PROGRAM AxisVertMovementOutputCtrl_Arm1
VAR
	VertTop: CMP_OC_DW;

	LdVertdown: CMP_OC_DW;
	Stn1Vertdown: CMP_OC_DW;
	Stn2Vertdown: CMP_OC_DW;
	Stn3Vertdown: CMP_OC_DW;
	Stn4Vertdown: CMP_OC_DW;
	Stn5Vertdown: CMP_OC_DW;
	Stn6Vertdown: CMP_OC_DW;
	Stn7Vertdown: CMP_OC_DW;
	Stn8Vertdown: CMP_OC_DW;
	Stn9Vertdown: CMP_OC_DW;
	Stn10Vertdown: CMP_OC_DW;
	Stn11Vertdown: CMP_OC_DW;
	Stn12Vertdown: CMP_OC_DW;
	Uld1Vertdown: CMP_OC_DW;
	Uld2Vertdown: CMP_OC_DW;

	Stn8VertSlowPulldown: CMP_OC_DW;

	Stn9VertSlowPulldown: CMP_OC_DW;
END_VAR

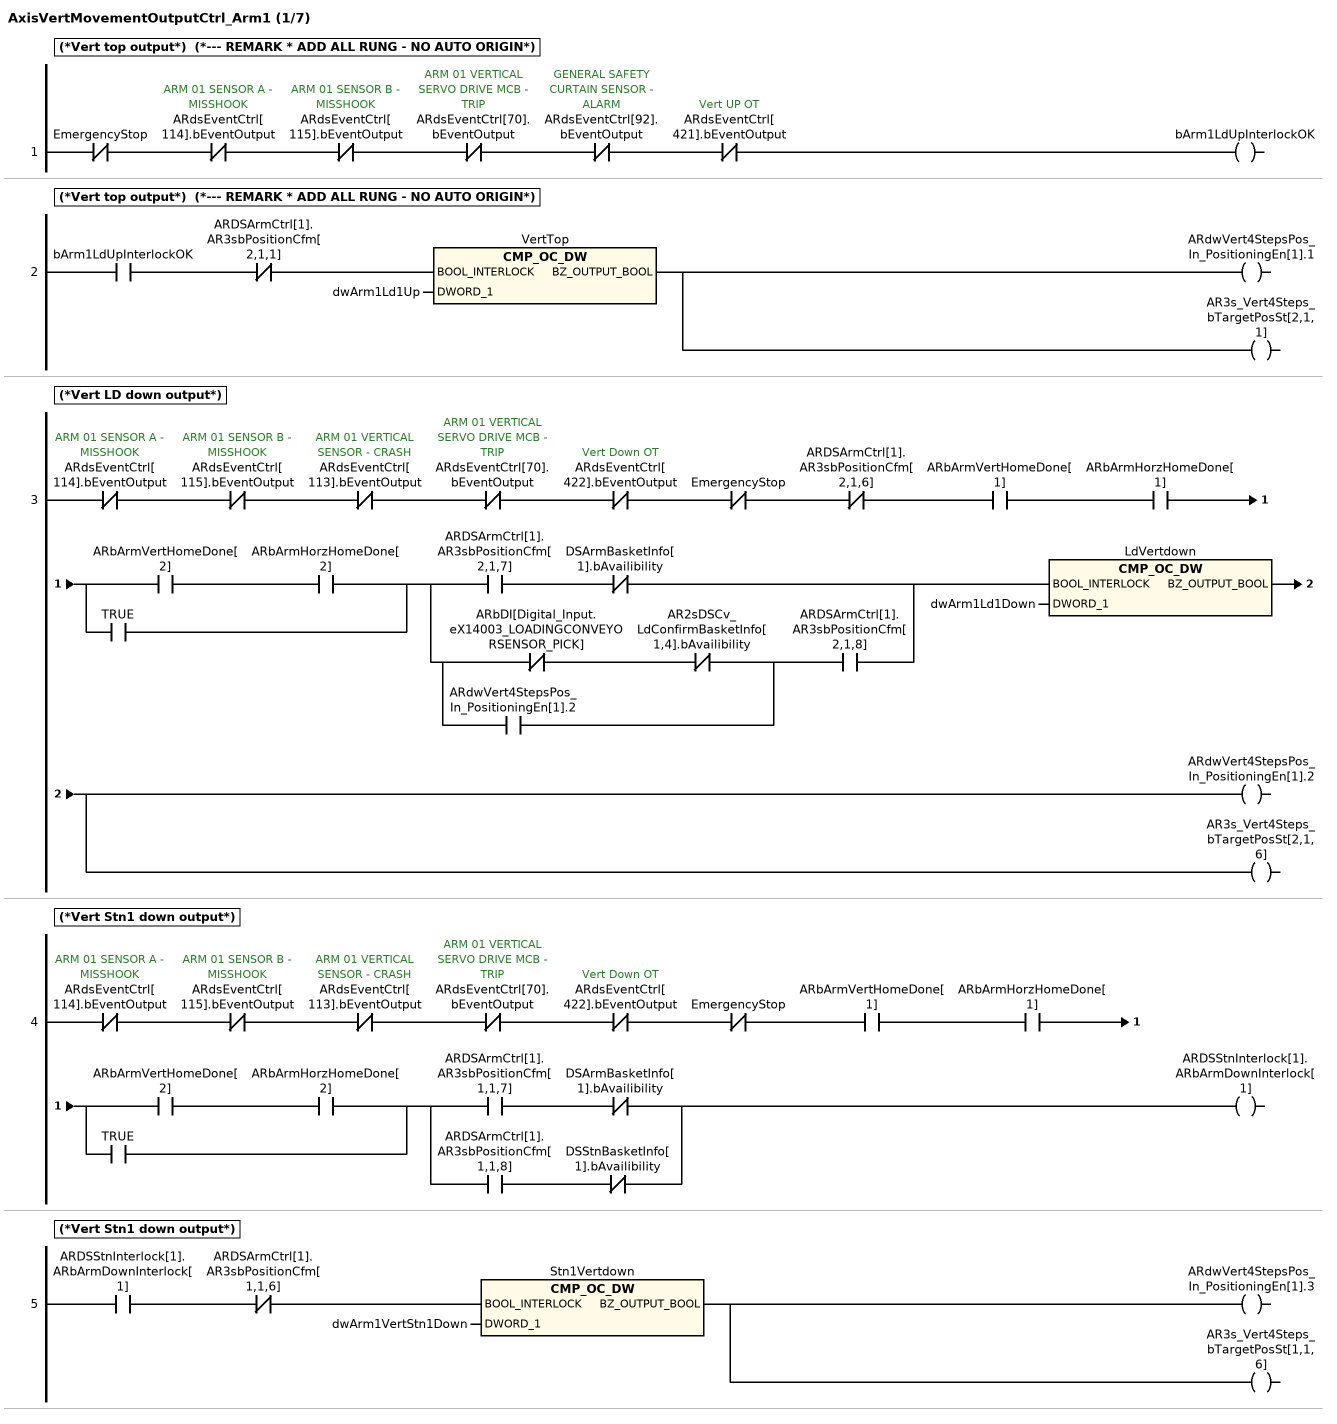
// NETWORK 1
//   ARdsEventCtrl[114].bEventOutput: ARM 01 SENSOR A - MISSHOOK
//   ARdsEventCtrl[115].bEventOutput: ARM 01 SENSOR B - MISSHOOK
//   ARdsEventCtrl[70].bEventOutput: ARM 01 VERTICAL SERVO DRIVE MCB - TRIP
//   ARdsEventCtrl[92].bEventOutput: GENERAL SAFETY CURTAIN SENSOR - ALARM
//   ARdsEventCtrl[421].bEventOutput: Vert UP OT
// label: (*Vert top output*)  (*--- REMARK * ADD ALL RUNG - NO AUTO ORIGIN*)
bArm1LdUpInterlockOK := NOT EmergencyStop AND NOT ARdsEventCtrl[114].bEventOutput AND NOT ARdsEventCtrl[115].bEventOutput AND NOT ARdsEventCtrl[70].bEventOutput AND NOT ARdsEventCtrl[92].bEventOutput AND NOT ARdsEventCtrl[421].bEventOutput;

// NETWORK 2
// label: (*Vert top output*)  (*--- REMARK * ADD ALL RUNG - NO AUTO ORIGIN*)
VertTop(BOOL_INTERLOCK := bArm1LdUpInterlockOK AND NOT ARDSArmCtrl[1].AR3sbPositionCfm[2,1,1], DWORD_1 := dwArm1Ld1Up); // CMP_OC_DW
ARdwVert4StepsPos_In_PositioningEn[1].1 := VertTop.BZ_OUTPUT_BOOL;
AR3s_Vert4Steps_bTargetPosSt[2,1,1] := VertTop.BZ_OUTPUT_BOOL;

// NETWORK 3
//   ARdsEventCtrl[114].bEventOutput: ARM 01 SENSOR A - MISSHOOK
//   ARdsEventCtrl[115].bEventOutput: ARM 01 SENSOR B - MISSHOOK
//   ARdsEventCtrl[113].bEventOutput: ARM 01 VERTICAL SENSOR - CRASH
//   ARdsEventCtrl[70].bEventOutput: ARM 01 VERTICAL SERVO DRIVE MCB - TRIP
//   ARdsEventCtrl[422].bEventOutput: Vert Down OT
// label: (*Vert LD down output*)
LdVertdown(BOOL_INTERLOCK := (NOT ARdsEventCtrl[114].bEventOutput AND NOT ARdsEventCtrl[115].bEventOutput AND NOT ARdsEventCtrl[113].bEventOutput AND NOT ARdsEventCtrl[70].bEventOutput AND NOT ARdsEventCtrl[422].bEventOutput AND NOT EmergencyStop) AND NOT ARDSArmCtrl[1].AR3sbPositionCfm[2,1,6] AND ARbArmVertHomeDone[1] AND ARbArmHorzHomeDone[1] AND (ARbArmVertHomeDone[2] AND ARbArmHorzHomeDone[2] OR TRUE) AND (ARDSArmCtrl[1].AR3sbPositionCfm[2,1,7] AND NOT DSArmBasketInfo[1].bAvailibility OR (NOT ARbDI[Digital_Input.eX14003_LOADINGCONVEYORSENSOR_PICK] AND NOT AR2sDSCv_LdConfirmBasketInfo[1,4].bAvailibility OR ARdwVert4StepsPos_In_PositioningEn[1].2) AND ARDSArmCtrl[1].AR3sbPositionCfm[2,1,8]), DWORD_1 := dwArm1Ld1Down); // CMP_OC_DW
ARdwVert4StepsPos_In_PositioningEn[1].2 := LdVertdown.BZ_OUTPUT_BOOL;
AR3s_Vert4Steps_bTargetPosSt[2,1,6] := LdVertdown.BZ_OUTPUT_BOOL;

// NETWORK 4
//   ARdsEventCtrl[114].bEventOutput: ARM 01 SENSOR A - MISSHOOK
//   ARdsEventCtrl[115].bEventOutput: ARM 01 SENSOR B - MISSHOOK
//   ARdsEventCtrl[113].bEventOutput: ARM 01 VERTICAL SENSOR - CRASH
//   ARdsEventCtrl[70].bEventOutput: ARM 01 VERTICAL SERVO DRIVE MCB - TRIP
//   ARdsEventCtrl[422].bEventOutput: Vert Down OT
// label: (*Vert Stn1 down output*)
ARDSStnInterlock[1].ARbArmDownInterlock[1] := (NOT ARdsEventCtrl[114].bEventOutput AND NOT ARdsEventCtrl[115].bEventOutput AND NOT ARdsEventCtrl[113].bEventOutput AND NOT ARdsEventCtrl[70].bEventOutput AND NOT ARdsEventCtrl[422].bEventOutput AND NOT EmergencyStop) AND ARbArmVertHomeDone[1] AND ARbArmHorzHomeDone[1] AND (ARbArmVertHomeDone[2] AND ARbArmHorzHomeDone[2] OR TRUE) AND (ARDSArmCtrl[1].AR3sbPositionCfm[1,1,7] AND NOT DSArmBasketInfo[1].bAvailibility OR ARDSArmCtrl[1].AR3sbPositionCfm[1,1,8] AND NOT DSStnBasketInfo[1].bAvailibility);

// NETWORK 5
// label: (*Vert Stn1 down output*)
Stn1Vertdown(BOOL_INTERLOCK := ARDSStnInterlock[1].ARbArmDownInterlock[1] AND NOT ARDSArmCtrl[1].AR3sbPositionCfm[1,1,6], DWORD_1 := dwArm1VertStn1Down); // CMP_OC_DW
ARdwVert4StepsPos_In_PositioningEn[1].3 := Stn1Vertdown.BZ_OUTPUT_BOOL;
AR3s_Vert4Steps_bTargetPosSt[1,1,6] := Stn1Vertdown.BZ_OUTPUT_BOOL;

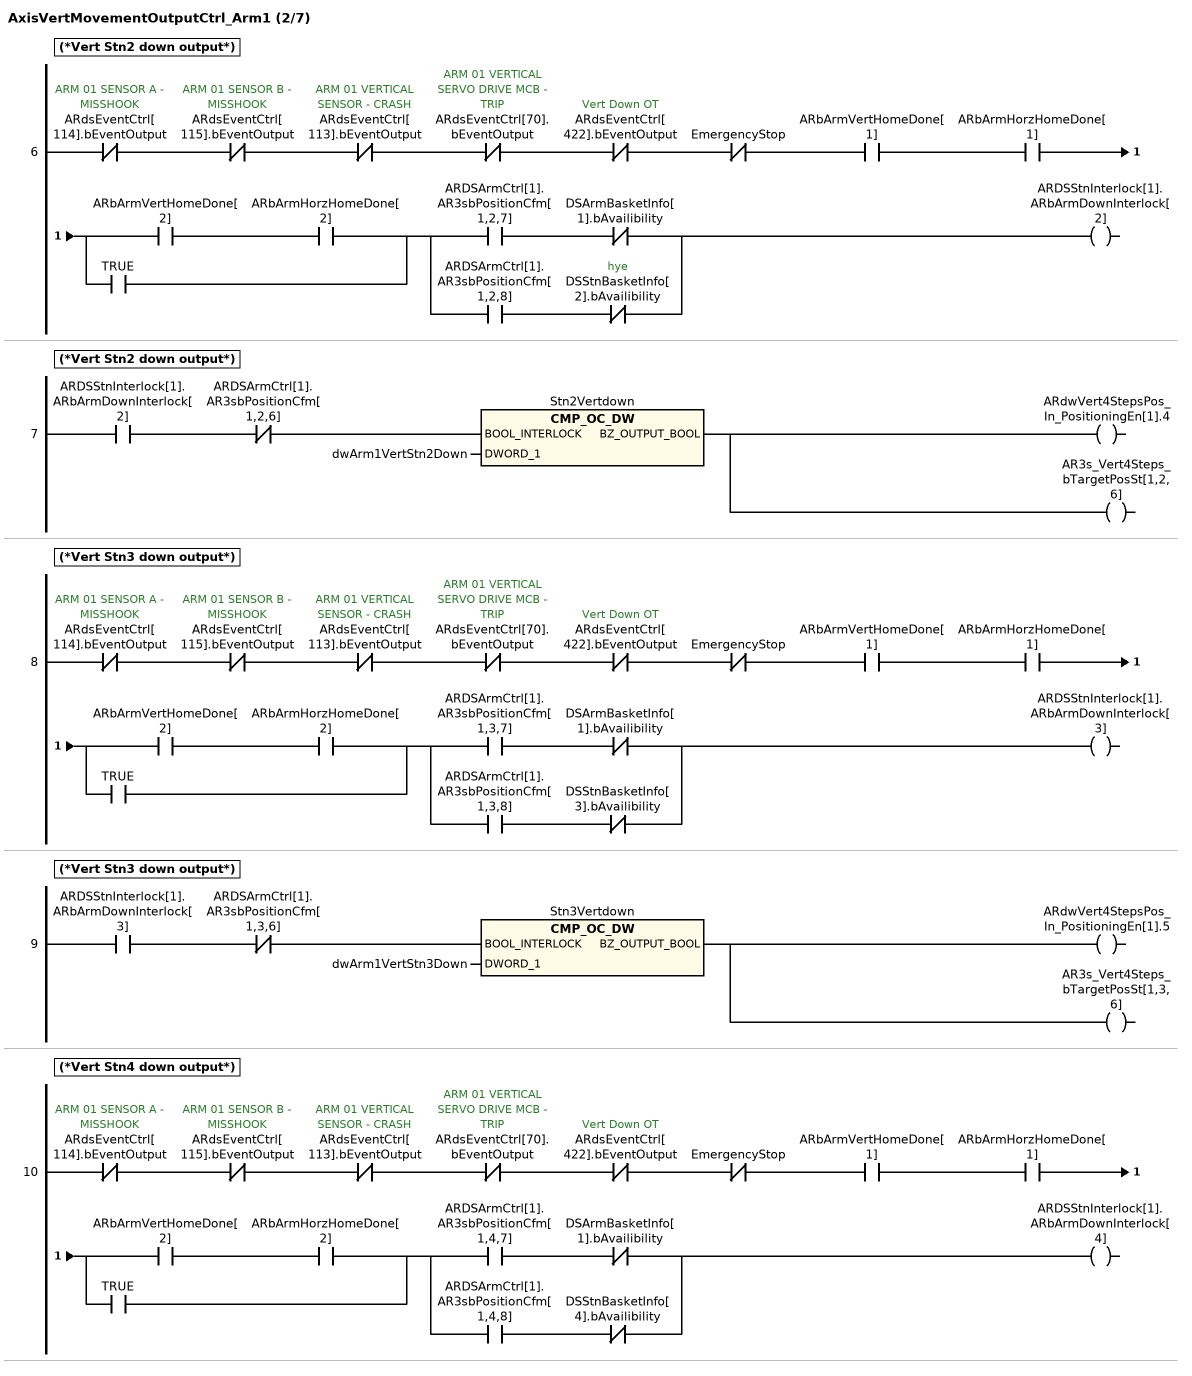
// NETWORK 6
//   ARdsEventCtrl[114].bEventOutput: ARM 01 SENSOR A - MISSHOOK
//   ARdsEventCtrl[115].bEventOutput: ARM 01 SENSOR B - MISSHOOK
//   ARdsEventCtrl[113].bEventOutput: ARM 01 VERTICAL SENSOR - CRASH
//   ARdsEventCtrl[70].bEventOutput: ARM 01 VERTICAL SERVO DRIVE MCB - TRIP
//   ARdsEventCtrl[422].bEventOutput: Vert Down OT
//   DSStnBasketInfo[2].bAvailibility: hye
// label: (*Vert Stn2 down output*)
ARDSStnInterlock[1].ARbArmDownInterlock[2] := (NOT ARdsEventCtrl[114].bEventOutput AND NOT ARdsEventCtrl[115].bEventOutput AND NOT ARdsEventCtrl[113].bEventOutput AND NOT ARdsEventCtrl[70].bEventOutput AND NOT ARdsEventCtrl[422].bEventOutput AND NOT EmergencyStop) AND ARbArmVertHomeDone[1] AND ARbArmHorzHomeDone[1] AND (ARbArmVertHomeDone[2] AND ARbArmHorzHomeDone[2] OR TRUE) AND (ARDSArmCtrl[1].AR3sbPositionCfm[1,2,7] AND NOT DSArmBasketInfo[1].bAvailibility OR ARDSArmCtrl[1].AR3sbPositionCfm[1,2,8] AND NOT DSStnBasketInfo[2].bAvailibility);

// NETWORK 7
// label: (*Vert Stn2 down output*)
Stn2Vertdown(BOOL_INTERLOCK := ARDSStnInterlock[1].ARbArmDownInterlock[2] AND NOT ARDSArmCtrl[1].AR3sbPositionCfm[1,2,6], DWORD_1 := dwArm1VertStn2Down); // CMP_OC_DW
ARdwVert4StepsPos_In_PositioningEn[1].4 := Stn2Vertdown.BZ_OUTPUT_BOOL;
AR3s_Vert4Steps_bTargetPosSt[1,2,6] := Stn2Vertdown.BZ_OUTPUT_BOOL;

// NETWORK 8
//   ARdsEventCtrl[114].bEventOutput: ARM 01 SENSOR A - MISSHOOK
//   ARdsEventCtrl[115].bEventOutput: ARM 01 SENSOR B - MISSHOOK
//   ARdsEventCtrl[113].bEventOutput: ARM 01 VERTICAL SENSOR - CRASH
//   ARdsEventCtrl[70].bEventOutput: ARM 01 VERTICAL SERVO DRIVE MCB - TRIP
//   ARdsEventCtrl[422].bEventOutput: Vert Down OT
// label: (*Vert Stn3 down output*)
ARDSStnInterlock[1].ARbArmDownInterlock[3] := (NOT ARdsEventCtrl[114].bEventOutput AND NOT ARdsEventCtrl[115].bEventOutput AND NOT ARdsEventCtrl[113].bEventOutput AND NOT ARdsEventCtrl[70].bEventOutput AND NOT ARdsEventCtrl[422].bEventOutput AND NOT EmergencyStop) AND ARbArmVertHomeDone[1] AND ARbArmHorzHomeDone[1] AND (ARbArmVertHomeDone[2] AND ARbArmHorzHomeDone[2] OR TRUE) AND (ARDSArmCtrl[1].AR3sbPositionCfm[1,3,7] AND NOT DSArmBasketInfo[1].bAvailibility OR ARDSArmCtrl[1].AR3sbPositionCfm[1,3,8] AND NOT DSStnBasketInfo[3].bAvailibility);

// NETWORK 9
// label: (*Vert Stn3 down output*)
Stn3Vertdown(BOOL_INTERLOCK := ARDSStnInterlock[1].ARbArmDownInterlock[3] AND NOT ARDSArmCtrl[1].AR3sbPositionCfm[1,3,6], DWORD_1 := dwArm1VertStn3Down); // CMP_OC_DW
ARdwVert4StepsPos_In_PositioningEn[1].5 := Stn3Vertdown.BZ_OUTPUT_BOOL;
AR3s_Vert4Steps_bTargetPosSt[1,3,6] := Stn3Vertdown.BZ_OUTPUT_BOOL;

// NETWORK 10
//   ARdsEventCtrl[114].bEventOutput: ARM 01 SENSOR A - MISSHOOK
//   ARdsEventCtrl[115].bEventOutput: ARM 01 SENSOR B - MISSHOOK
//   ARdsEventCtrl[113].bEventOutput: ARM 01 VERTICAL SENSOR - CRASH
//   ARdsEventCtrl[70].bEventOutput: ARM 01 VERTICAL SERVO DRIVE MCB - TRIP
//   ARdsEventCtrl[422].bEventOutput: Vert Down OT
// label: (*Vert Stn4 down output*)
ARDSStnInterlock[1].ARbArmDownInterlock[4] := (NOT ARdsEventCtrl[114].bEventOutput AND NOT ARdsEventCtrl[115].bEventOutput AND NOT ARdsEventCtrl[113].bEventOutput AND NOT ARdsEventCtrl[70].bEventOutput AND NOT ARdsEventCtrl[422].bEventOutput AND NOT EmergencyStop) AND ARbArmVertHomeDone[1] AND ARbArmHorzHomeDone[1] AND (ARbArmVertHomeDone[2] AND ARbArmHorzHomeDone[2] OR TRUE) AND (ARDSArmCtrl[1].AR3sbPositionCfm[1,4,7] AND NOT DSArmBasketInfo[1].bAvailibility OR ARDSArmCtrl[1].AR3sbPositionCfm[1,4,8] AND NOT DSStnBasketInfo[4].bAvailibility);

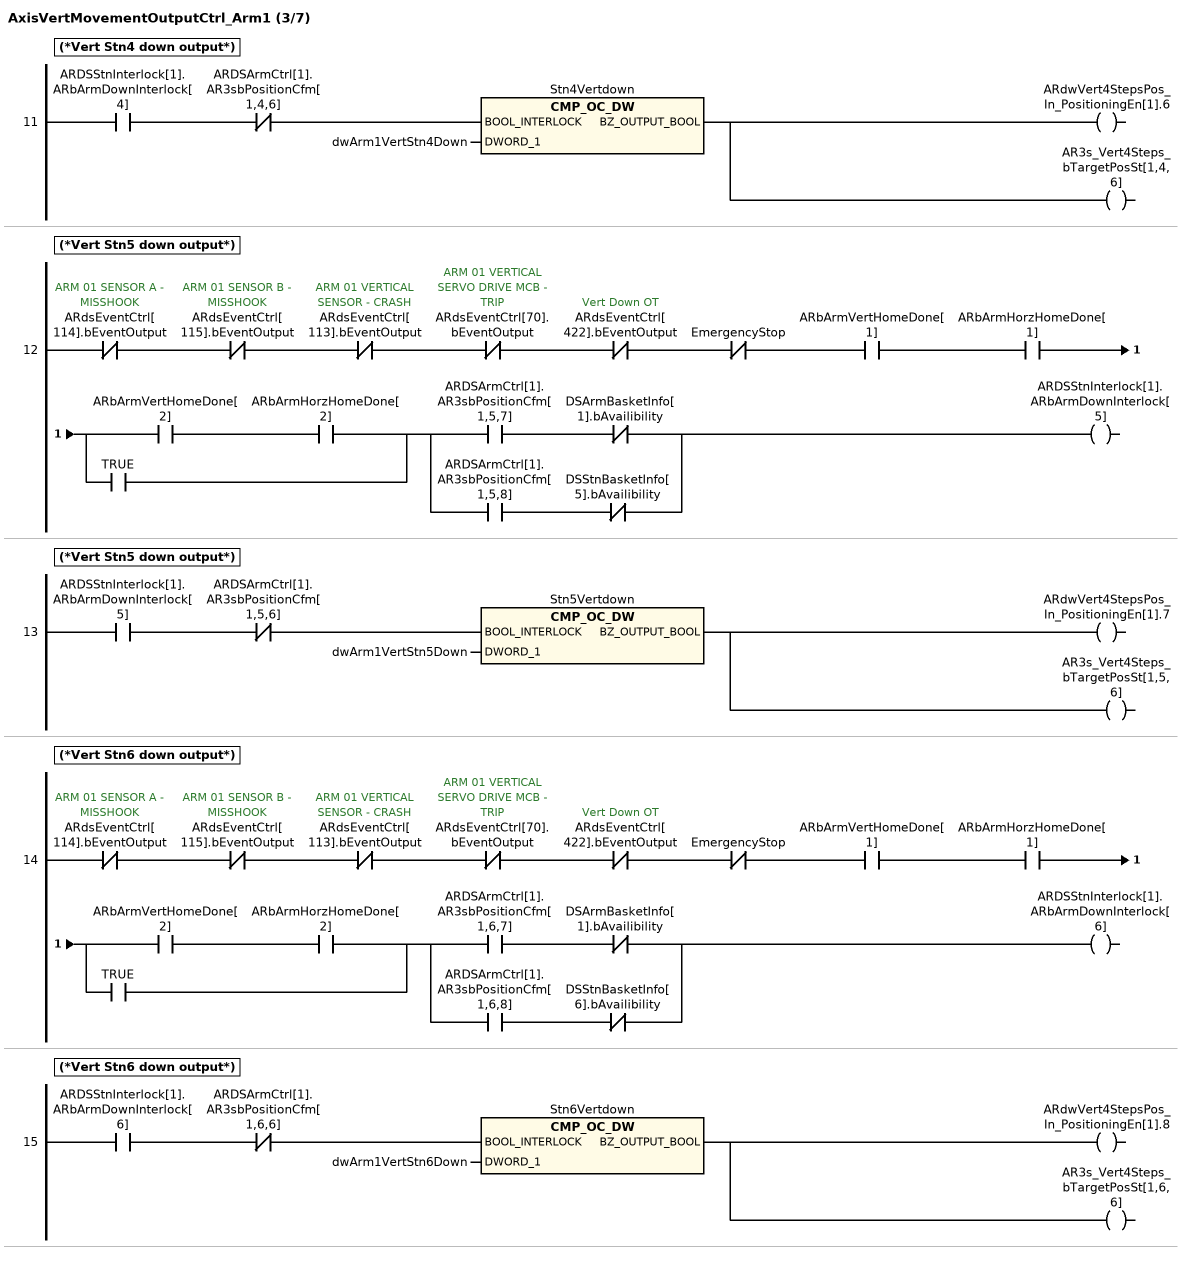
// NETWORK 11
// label: (*Vert Stn4 down output*)
Stn4Vertdown(BOOL_INTERLOCK := ARDSStnInterlock[1].ARbArmDownInterlock[4] AND NOT ARDSArmCtrl[1].AR3sbPositionCfm[1,4,6], DWORD_1 := dwArm1VertStn4Down); // CMP_OC_DW
ARdwVert4StepsPos_In_PositioningEn[1].6 := Stn4Vertdown.BZ_OUTPUT_BOOL;
AR3s_Vert4Steps_bTargetPosSt[1,4,6] := Stn4Vertdown.BZ_OUTPUT_BOOL;

// NETWORK 12
//   ARdsEventCtrl[114].bEventOutput: ARM 01 SENSOR A - MISSHOOK
//   ARdsEventCtrl[115].bEventOutput: ARM 01 SENSOR B - MISSHOOK
//   ARdsEventCtrl[113].bEventOutput: ARM 01 VERTICAL SENSOR - CRASH
//   ARdsEventCtrl[70].bEventOutput: ARM 01 VERTICAL SERVO DRIVE MCB - TRIP
//   ARdsEventCtrl[422].bEventOutput: Vert Down OT
// label: (*Vert Stn5 down output*)
ARDSStnInterlock[1].ARbArmDownInterlock[5] := (NOT ARdsEventCtrl[114].bEventOutput AND NOT ARdsEventCtrl[115].bEventOutput AND NOT ARdsEventCtrl[113].bEventOutput AND NOT ARdsEventCtrl[70].bEventOutput AND NOT ARdsEventCtrl[422].bEventOutput AND NOT EmergencyStop) AND ARbArmVertHomeDone[1] AND ARbArmHorzHomeDone[1] AND (ARbArmVertHomeDone[2] AND ARbArmHorzHomeDone[2] OR TRUE) AND (ARDSArmCtrl[1].AR3sbPositionCfm[1,5,7] AND NOT DSArmBasketInfo[1].bAvailibility OR ARDSArmCtrl[1].AR3sbPositionCfm[1,5,8] AND NOT DSStnBasketInfo[5].bAvailibility);

// NETWORK 13
// label: (*Vert Stn5 down output*)
Stn5Vertdown(BOOL_INTERLOCK := ARDSStnInterlock[1].ARbArmDownInterlock[5] AND NOT ARDSArmCtrl[1].AR3sbPositionCfm[1,5,6], DWORD_1 := dwArm1VertStn5Down); // CMP_OC_DW
ARdwVert4StepsPos_In_PositioningEn[1].7 := Stn5Vertdown.BZ_OUTPUT_BOOL;
AR3s_Vert4Steps_bTargetPosSt[1,5,6] := Stn5Vertdown.BZ_OUTPUT_BOOL;

// NETWORK 14
//   ARdsEventCtrl[114].bEventOutput: ARM 01 SENSOR A - MISSHOOK
//   ARdsEventCtrl[115].bEventOutput: ARM 01 SENSOR B - MISSHOOK
//   ARdsEventCtrl[113].bEventOutput: ARM 01 VERTICAL SENSOR - CRASH
//   ARdsEventCtrl[70].bEventOutput: ARM 01 VERTICAL SERVO DRIVE MCB - TRIP
//   ARdsEventCtrl[422].bEventOutput: Vert Down OT
// label: (*Vert Stn6 down output*)
ARDSStnInterlock[1].ARbArmDownInterlock[6] := (NOT ARdsEventCtrl[114].bEventOutput AND NOT ARdsEventCtrl[115].bEventOutput AND NOT ARdsEventCtrl[113].bEventOutput AND NOT ARdsEventCtrl[70].bEventOutput AND NOT ARdsEventCtrl[422].bEventOutput AND NOT EmergencyStop) AND ARbArmVertHomeDone[1] AND ARbArmHorzHomeDone[1] AND (ARbArmVertHomeDone[2] AND ARbArmHorzHomeDone[2] OR TRUE) AND (ARDSArmCtrl[1].AR3sbPositionCfm[1,6,7] AND NOT DSArmBasketInfo[1].bAvailibility OR ARDSArmCtrl[1].AR3sbPositionCfm[1,6,8] AND NOT DSStnBasketInfo[6].bAvailibility);

// NETWORK 15
// label: (*Vert Stn6 down output*)
Stn6Vertdown(BOOL_INTERLOCK := ARDSStnInterlock[1].ARbArmDownInterlock[6] AND NOT ARDSArmCtrl[1].AR3sbPositionCfm[1,6,6], DWORD_1 := dwArm1VertStn6Down); // CMP_OC_DW
ARdwVert4StepsPos_In_PositioningEn[1].8 := Stn6Vertdown.BZ_OUTPUT_BOOL;
AR3s_Vert4Steps_bTargetPosSt[1,6,6] := Stn6Vertdown.BZ_OUTPUT_BOOL;

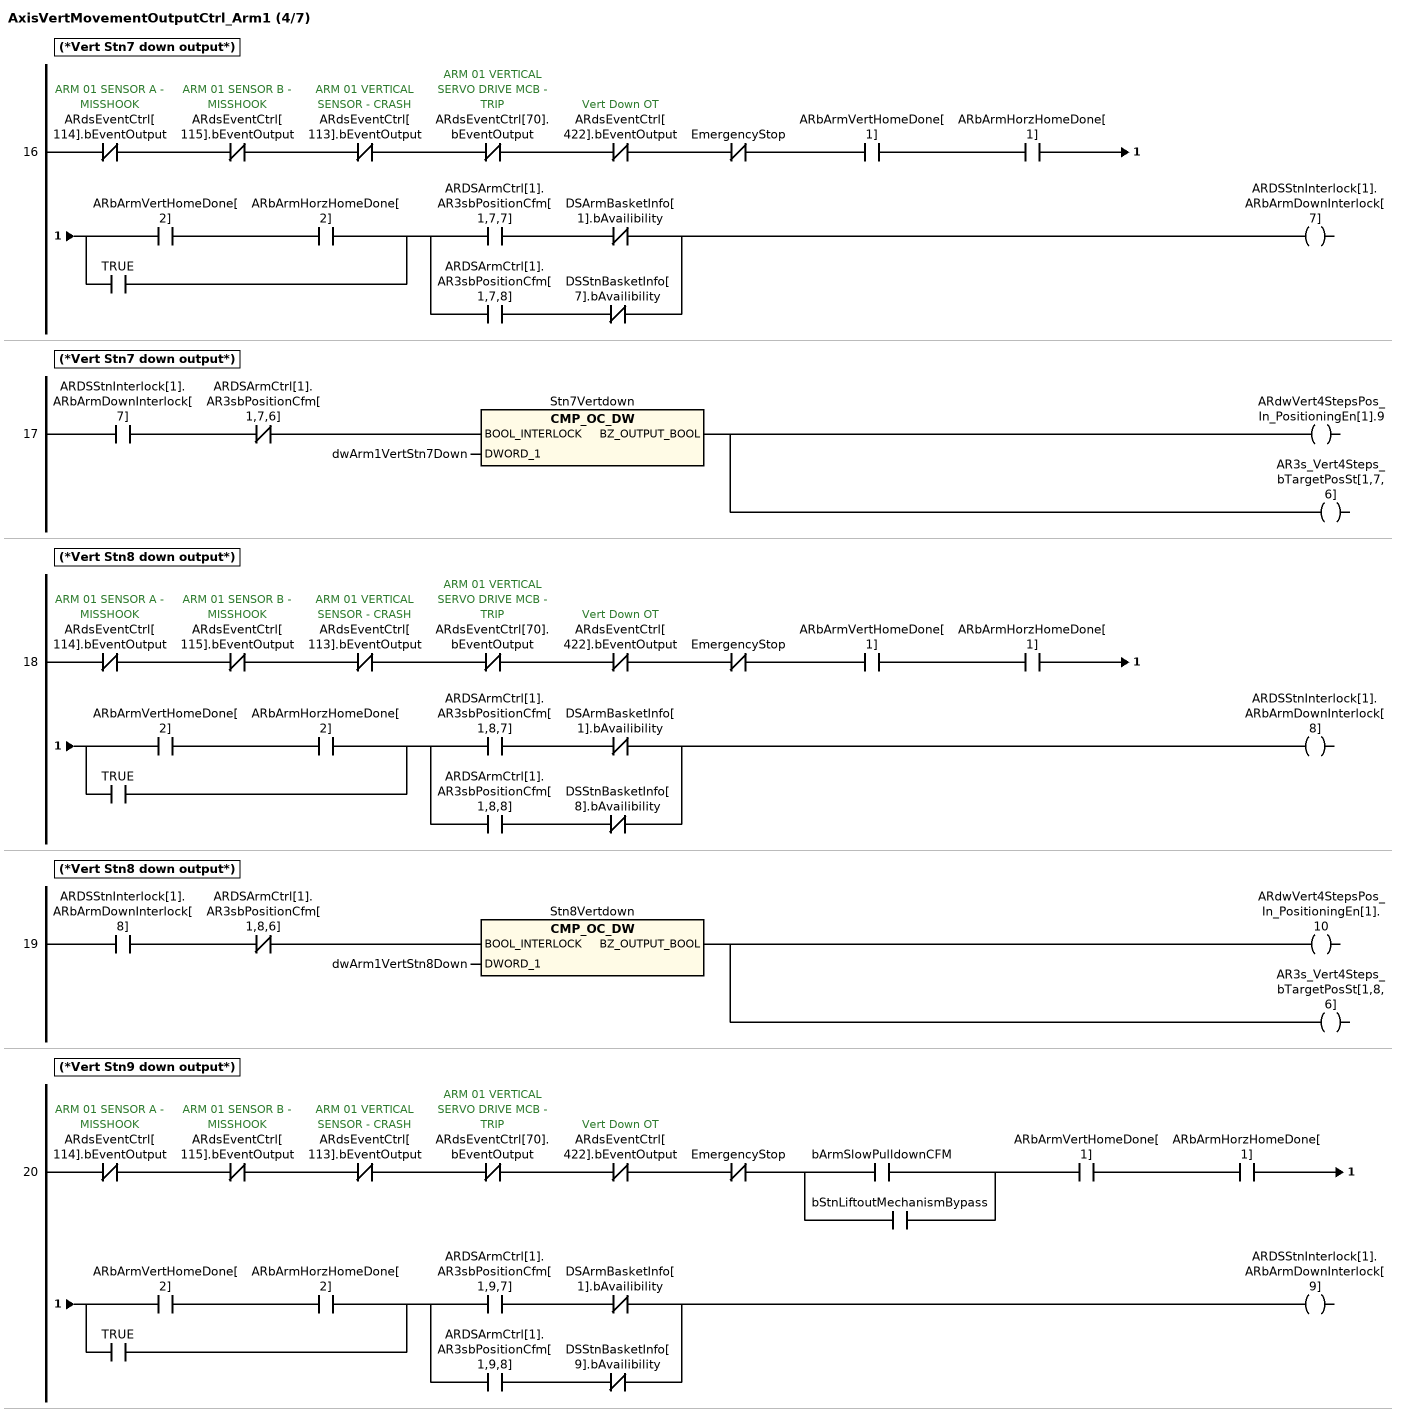
// NETWORK 16
//   ARdsEventCtrl[114].bEventOutput: ARM 01 SENSOR A - MISSHOOK
//   ARdsEventCtrl[115].bEventOutput: ARM 01 SENSOR B - MISSHOOK
//   ARdsEventCtrl[113].bEventOutput: ARM 01 VERTICAL SENSOR - CRASH
//   ARdsEventCtrl[70].bEventOutput: ARM 01 VERTICAL SERVO DRIVE MCB - TRIP
//   ARdsEventCtrl[422].bEventOutput: Vert Down OT
// label: (*Vert Stn7 down output*)
ARDSStnInterlock[1].ARbArmDownInterlock[7] := (NOT ARdsEventCtrl[114].bEventOutput AND NOT ARdsEventCtrl[115].bEventOutput AND NOT ARdsEventCtrl[113].bEventOutput AND NOT ARdsEventCtrl[70].bEventOutput AND NOT ARdsEventCtrl[422].bEventOutput AND NOT EmergencyStop) AND ARbArmVertHomeDone[1] AND ARbArmHorzHomeDone[1] AND (ARbArmVertHomeDone[2] AND ARbArmHorzHomeDone[2] OR TRUE) AND (ARDSArmCtrl[1].AR3sbPositionCfm[1,7,7] AND NOT DSArmBasketInfo[1].bAvailibility OR ARDSArmCtrl[1].AR3sbPositionCfm[1,7,8] AND NOT DSStnBasketInfo[7].bAvailibility);

// NETWORK 17
// label: (*Vert Stn7 down output*)
Stn7Vertdown(BOOL_INTERLOCK := ARDSStnInterlock[1].ARbArmDownInterlock[7] AND NOT ARDSArmCtrl[1].AR3sbPositionCfm[1,7,6], DWORD_1 := dwArm1VertStn7Down); // CMP_OC_DW
ARdwVert4StepsPos_In_PositioningEn[1].9 := Stn7Vertdown.BZ_OUTPUT_BOOL;
AR3s_Vert4Steps_bTargetPosSt[1,7,6] := Stn7Vertdown.BZ_OUTPUT_BOOL;

// NETWORK 18
//   ARdsEventCtrl[114].bEventOutput: ARM 01 SENSOR A - MISSHOOK
//   ARdsEventCtrl[115].bEventOutput: ARM 01 SENSOR B - MISSHOOK
//   ARdsEventCtrl[113].bEventOutput: ARM 01 VERTICAL SENSOR - CRASH
//   ARdsEventCtrl[70].bEventOutput: ARM 01 VERTICAL SERVO DRIVE MCB - TRIP
//   ARdsEventCtrl[422].bEventOutput: Vert Down OT
// label: (*Vert Stn8 down output*)
ARDSStnInterlock[1].ARbArmDownInterlock[8] := (NOT ARdsEventCtrl[114].bEventOutput AND NOT ARdsEventCtrl[115].bEventOutput AND NOT ARdsEventCtrl[113].bEventOutput AND NOT ARdsEventCtrl[70].bEventOutput AND NOT ARdsEventCtrl[422].bEventOutput AND NOT EmergencyStop) AND ARbArmVertHomeDone[1] AND ARbArmHorzHomeDone[1] AND (ARbArmVertHomeDone[2] AND ARbArmHorzHomeDone[2] OR TRUE) AND (ARDSArmCtrl[1].AR3sbPositionCfm[1,8,7] AND NOT DSArmBasketInfo[1].bAvailibility OR ARDSArmCtrl[1].AR3sbPositionCfm[1,8,8] AND NOT DSStnBasketInfo[8].bAvailibility);

// NETWORK 19
// label: (*Vert Stn8 down output*)
Stn8Vertdown(BOOL_INTERLOCK := ARDSStnInterlock[1].ARbArmDownInterlock[8] AND NOT ARDSArmCtrl[1].AR3sbPositionCfm[1,8,6], DWORD_1 := dwArm1VertStn8Down); // CMP_OC_DW
ARdwVert4StepsPos_In_PositioningEn[1].10 := Stn8Vertdown.BZ_OUTPUT_BOOL;
AR3s_Vert4Steps_bTargetPosSt[1,8,6] := Stn8Vertdown.BZ_OUTPUT_BOOL;

// NETWORK 20
//   ARdsEventCtrl[114].bEventOutput: ARM 01 SENSOR A - MISSHOOK
//   ARdsEventCtrl[115].bEventOutput: ARM 01 SENSOR B - MISSHOOK
//   ARdsEventCtrl[113].bEventOutput: ARM 01 VERTICAL SENSOR - CRASH
//   ARdsEventCtrl[70].bEventOutput: ARM 01 VERTICAL SERVO DRIVE MCB - TRIP
//   ARdsEventCtrl[422].bEventOutput: Vert Down OT
// label: (*Vert Stn9 down output*)
ARDSStnInterlock[1].ARbArmDownInterlock[9] := (NOT ARdsEventCtrl[114].bEventOutput AND NOT ARdsEventCtrl[115].bEventOutput AND NOT ARdsEventCtrl[113].bEventOutput AND NOT ARdsEventCtrl[70].bEventOutput AND NOT ARdsEventCtrl[422].bEventOutput AND NOT EmergencyStop AND (bArmSlowPulldownCFM OR bStnLiftoutMechanismBypass)) AND ARbArmVertHomeDone[1] AND ARbArmHorzHomeDone[1] AND (ARbArmVertHomeDone[2] AND ARbArmHorzHomeDone[2] OR TRUE) AND (ARDSArmCtrl[1].AR3sbPositionCfm[1,9,7] AND NOT DSArmBasketInfo[1].bAvailibility OR ARDSArmCtrl[1].AR3sbPositionCfm[1,9,8] AND NOT DSStnBasketInfo[9].bAvailibility);

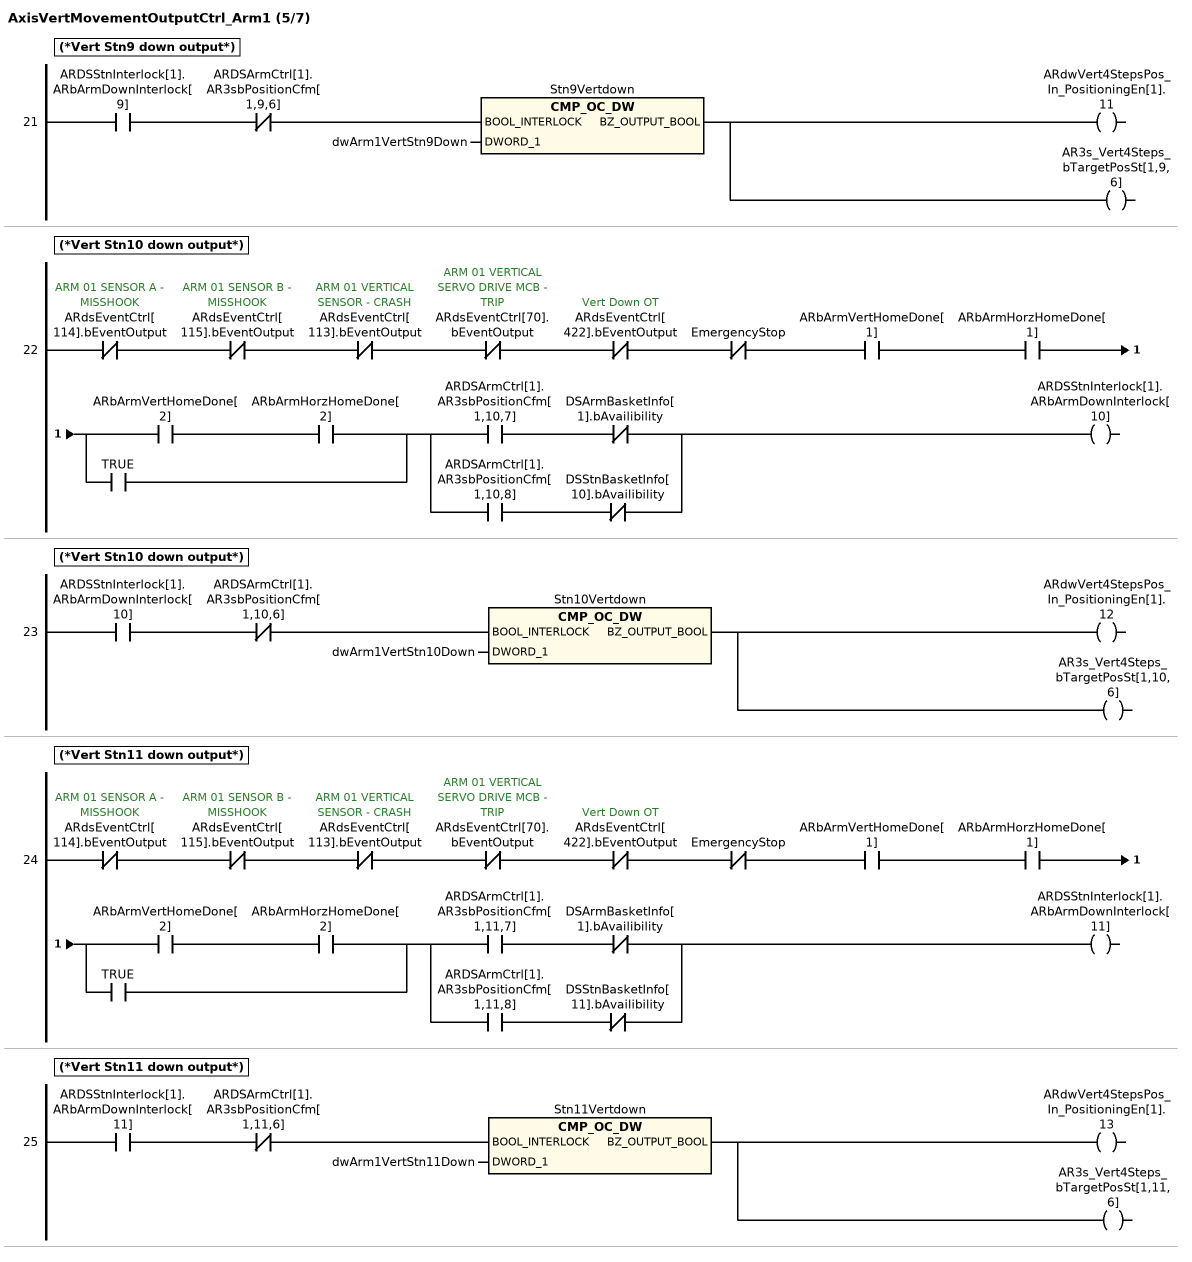
// NETWORK 21
// label: (*Vert Stn9 down output*)
Stn9Vertdown(BOOL_INTERLOCK := ARDSStnInterlock[1].ARbArmDownInterlock[9] AND NOT ARDSArmCtrl[1].AR3sbPositionCfm[1,9,6], DWORD_1 := dwArm1VertStn9Down); // CMP_OC_DW
ARdwVert4StepsPos_In_PositioningEn[1].11 := Stn9Vertdown.BZ_OUTPUT_BOOL;
AR3s_Vert4Steps_bTargetPosSt[1,9,6] := Stn9Vertdown.BZ_OUTPUT_BOOL;

// NETWORK 22
//   ARdsEventCtrl[114].bEventOutput: ARM 01 SENSOR A - MISSHOOK
//   ARdsEventCtrl[115].bEventOutput: ARM 01 SENSOR B - MISSHOOK
//   ARdsEventCtrl[113].bEventOutput: ARM 01 VERTICAL SENSOR - CRASH
//   ARdsEventCtrl[70].bEventOutput: ARM 01 VERTICAL SERVO DRIVE MCB - TRIP
//   ARdsEventCtrl[422].bEventOutput: Vert Down OT
// label: (*Vert Stn10 down output*)
ARDSStnInterlock[1].ARbArmDownInterlock[10] := (NOT ARdsEventCtrl[114].bEventOutput AND NOT ARdsEventCtrl[115].bEventOutput AND NOT ARdsEventCtrl[113].bEventOutput AND NOT ARdsEventCtrl[70].bEventOutput AND NOT ARdsEventCtrl[422].bEventOutput AND NOT EmergencyStop) AND ARbArmVertHomeDone[1] AND ARbArmHorzHomeDone[1] AND (ARbArmVertHomeDone[2] AND ARbArmHorzHomeDone[2] OR TRUE) AND (ARDSArmCtrl[1].AR3sbPositionCfm[1,10,7] AND NOT DSArmBasketInfo[1].bAvailibility OR ARDSArmCtrl[1].AR3sbPositionCfm[1,10,8] AND NOT DSStnBasketInfo[10].bAvailibility);

// NETWORK 23
// label: (*Vert Stn10 down output*)
Stn10Vertdown(BOOL_INTERLOCK := ARDSStnInterlock[1].ARbArmDownInterlock[10] AND NOT ARDSArmCtrl[1].AR3sbPositionCfm[1,10,6], DWORD_1 := dwArm1VertStn10Down); // CMP_OC_DW
ARdwVert4StepsPos_In_PositioningEn[1].12 := Stn10Vertdown.BZ_OUTPUT_BOOL;
AR3s_Vert4Steps_bTargetPosSt[1,10,6] := Stn10Vertdown.BZ_OUTPUT_BOOL;

// NETWORK 24
//   ARdsEventCtrl[114].bEventOutput: ARM 01 SENSOR A - MISSHOOK
//   ARdsEventCtrl[115].bEventOutput: ARM 01 SENSOR B - MISSHOOK
//   ARdsEventCtrl[113].bEventOutput: ARM 01 VERTICAL SENSOR - CRASH
//   ARdsEventCtrl[70].bEventOutput: ARM 01 VERTICAL SERVO DRIVE MCB - TRIP
//   ARdsEventCtrl[422].bEventOutput: Vert Down OT
// label: (*Vert Stn11 down output*)
ARDSStnInterlock[1].ARbArmDownInterlock[11] := (NOT ARdsEventCtrl[114].bEventOutput AND NOT ARdsEventCtrl[115].bEventOutput AND NOT ARdsEventCtrl[113].bEventOutput AND NOT ARdsEventCtrl[70].bEventOutput AND NOT ARdsEventCtrl[422].bEventOutput AND NOT EmergencyStop) AND ARbArmVertHomeDone[1] AND ARbArmHorzHomeDone[1] AND (ARbArmVertHomeDone[2] AND ARbArmHorzHomeDone[2] OR TRUE) AND (ARDSArmCtrl[1].AR3sbPositionCfm[1,11,7] AND NOT DSArmBasketInfo[1].bAvailibility OR ARDSArmCtrl[1].AR3sbPositionCfm[1,11,8] AND NOT DSStnBasketInfo[11].bAvailibility);

// NETWORK 25
// label: (*Vert Stn11 down output*)
Stn11Vertdown(BOOL_INTERLOCK := ARDSStnInterlock[1].ARbArmDownInterlock[11] AND NOT ARDSArmCtrl[1].AR3sbPositionCfm[1,11,6], DWORD_1 := dwArm1VertStn11Down); // CMP_OC_DW
ARdwVert4StepsPos_In_PositioningEn[1].13 := Stn11Vertdown.BZ_OUTPUT_BOOL;
AR3s_Vert4Steps_bTargetPosSt[1,11,6] := Stn11Vertdown.BZ_OUTPUT_BOOL;

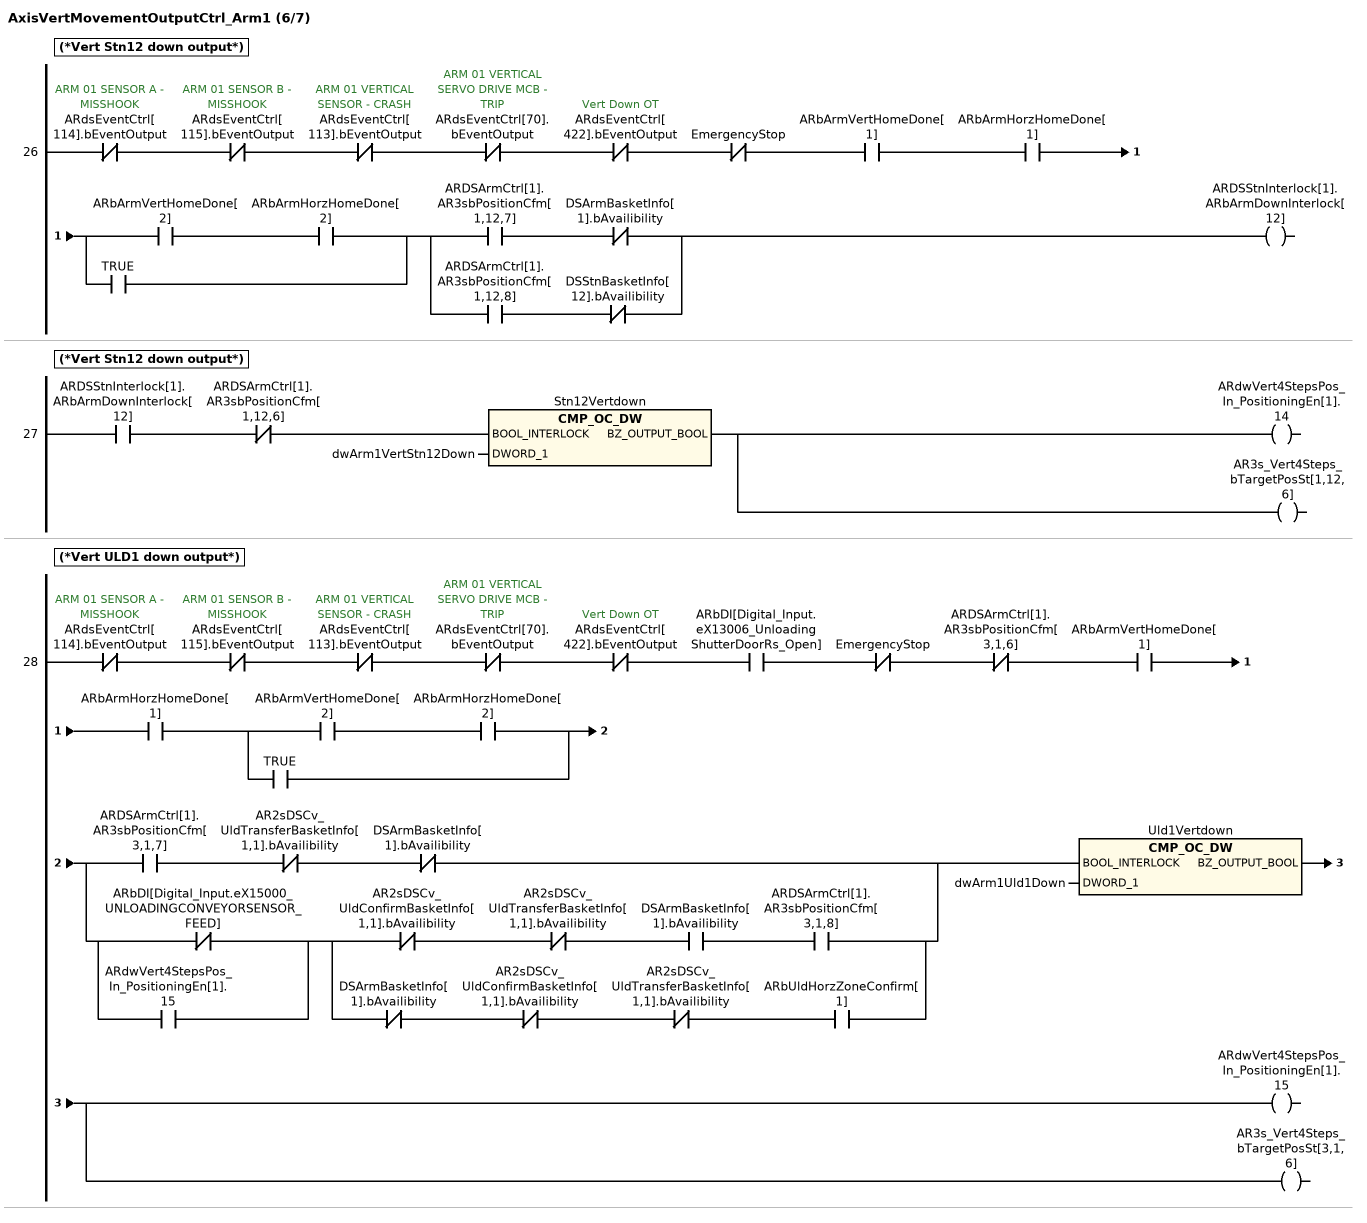
// NETWORK 26
//   ARdsEventCtrl[114].bEventOutput: ARM 01 SENSOR A - MISSHOOK
//   ARdsEventCtrl[115].bEventOutput: ARM 01 SENSOR B - MISSHOOK
//   ARdsEventCtrl[113].bEventOutput: ARM 01 VERTICAL SENSOR - CRASH
//   ARdsEventCtrl[70].bEventOutput: ARM 01 VERTICAL SERVO DRIVE MCB - TRIP
//   ARdsEventCtrl[422].bEventOutput: Vert Down OT
// label: (*Vert Stn12 down output*)
ARDSStnInterlock[1].ARbArmDownInterlock[12] := (NOT ARdsEventCtrl[114].bEventOutput AND NOT ARdsEventCtrl[115].bEventOutput AND NOT ARdsEventCtrl[113].bEventOutput AND NOT ARdsEventCtrl[70].bEventOutput AND NOT ARdsEventCtrl[422].bEventOutput AND NOT EmergencyStop) AND ARbArmVertHomeDone[1] AND ARbArmHorzHomeDone[1] AND (ARbArmVertHomeDone[2] AND ARbArmHorzHomeDone[2] OR TRUE) AND (ARDSArmCtrl[1].AR3sbPositionCfm[1,12,7] AND NOT DSArmBasketInfo[1].bAvailibility OR ARDSArmCtrl[1].AR3sbPositionCfm[1,12,8] AND NOT DSStnBasketInfo[12].bAvailibility);

// NETWORK 27
// label: (*Vert Stn12 down output*)
Stn12Vertdown(BOOL_INTERLOCK := ARDSStnInterlock[1].ARbArmDownInterlock[12] AND NOT ARDSArmCtrl[1].AR3sbPositionCfm[1,12,6], DWORD_1 := dwArm1VertStn12Down); // CMP_OC_DW
ARdwVert4StepsPos_In_PositioningEn[1].14 := Stn12Vertdown.BZ_OUTPUT_BOOL;
AR3s_Vert4Steps_bTargetPosSt[1,12,6] := Stn12Vertdown.BZ_OUTPUT_BOOL;

// NETWORK 28
//   ARdsEventCtrl[114].bEventOutput: ARM 01 SENSOR A - MISSHOOK
//   ARdsEventCtrl[115].bEventOutput: ARM 01 SENSOR B - MISSHOOK
//   ARdsEventCtrl[113].bEventOutput: ARM 01 VERTICAL SENSOR - CRASH
//   ARdsEventCtrl[70].bEventOutput: ARM 01 VERTICAL SERVO DRIVE MCB - TRIP
//   ARdsEventCtrl[422].bEventOutput: Vert Down OT
// label: (*Vert ULD1 down output*)
Uld1Vertdown(BOOL_INTERLOCK := (NOT ARdsEventCtrl[114].bEventOutput AND NOT ARdsEventCtrl[115].bEventOutput AND NOT ARdsEventCtrl[113].bEventOutput AND NOT ARdsEventCtrl[70].bEventOutput AND NOT ARdsEventCtrl[422].bEventOutput AND ARbDI[Digital_Input.eX13006_UnloadingShutterDoorRs_Open] AND NOT EmergencyStop) AND NOT ARDSArmCtrl[1].AR3sbPositionCfm[3,1,6] AND ARbArmVertHomeDone[1] AND ARbArmHorzHomeDone[1] AND (ARbArmVertHomeDone[2] AND ARbArmHorzHomeDone[2] OR TRUE) AND (ARDSArmCtrl[1].AR3sbPositionCfm[3,1,7] AND NOT AR2sDSCv_UldTransferBasketInfo[1,1].bAvailibility AND NOT DSArmBasketInfo[1].bAvailibility OR (NOT ARbDI[Digital_Input.eX15000_UNLOADINGCONVEYORSENSOR_FEED] OR ARdwVert4StepsPos_In_PositioningEn[1].15) AND (NOT AR2sDSCv_UldConfirmBasketInfo[1,1].bAvailibility AND NOT AR2sDSCv_UldTransferBasketInfo[1,1].bAvailibility AND DSArmBasketInfo[1].bAvailibility AND ARDSArmCtrl[1].AR3sbPositionCfm[3,1,8] OR NOT DSArmBasketInfo[1].bAvailibility AND NOT AR2sDSCv_UldConfirmBasketInfo[1,1].bAvailibility AND NOT AR2sDSCv_UldTransferBasketInfo[1,1].bAvailibility AND ARbUldHorzZoneConfirm[1])), DWORD_1 := dwArm1Uld1Down); // CMP_OC_DW
ARdwVert4StepsPos_In_PositioningEn[1].15 := Uld1Vertdown.BZ_OUTPUT_BOOL;
AR3s_Vert4Steps_bTargetPosSt[3,1,6] := Uld1Vertdown.BZ_OUTPUT_BOOL;

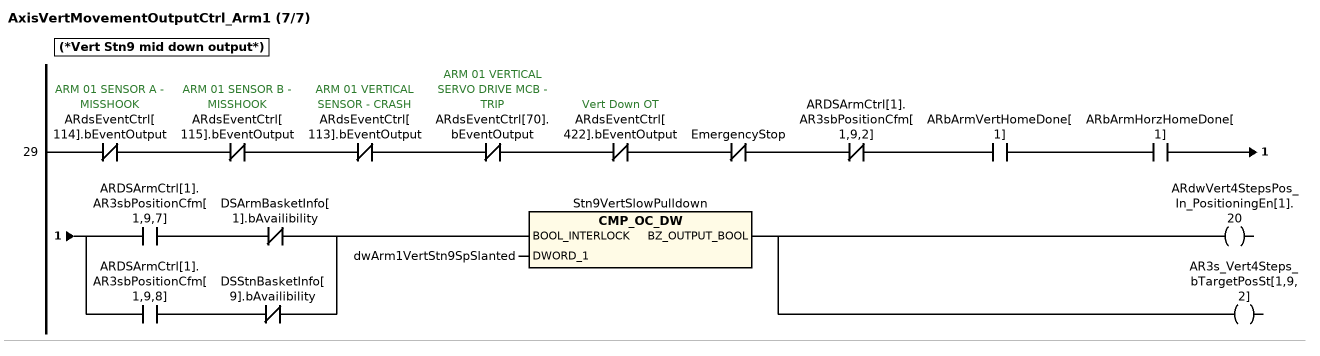
// NETWORK 29
//   ARdsEventCtrl[114].bEventOutput: ARM 01 SENSOR A - MISSHOOK
//   ARdsEventCtrl[115].bEventOutput: ARM 01 SENSOR B - MISSHOOK
//   ARdsEventCtrl[113].bEventOutput: ARM 01 VERTICAL SENSOR - CRASH
//   ARdsEventCtrl[70].bEventOutput: ARM 01 VERTICAL SERVO DRIVE MCB - TRIP
//   ARdsEventCtrl[422].bEventOutput: Vert Down OT
// label: (*Vert Stn9 mid down output*)
Stn9VertSlowPulldown(BOOL_INTERLOCK := (NOT ARdsEventCtrl[114].bEventOutput AND NOT ARdsEventCtrl[115].bEventOutput AND NOT ARdsEventCtrl[113].bEventOutput AND NOT ARdsEventCtrl[70].bEventOutput AND NOT ARdsEventCtrl[422].bEventOutput AND NOT EmergencyStop) AND NOT ARDSArmCtrl[1].AR3sbPositionCfm[1,9,2] AND ARbArmVertHomeDone[1] AND ARbArmHorzHomeDone[1] AND (ARDSArmCtrl[1].AR3sbPositionCfm[1,9,7] AND NOT DSArmBasketInfo[1].bAvailibility OR ARDSArmCtrl[1].AR3sbPositionCfm[1,9,8] AND NOT DSStnBasketInfo[9].bAvailibility), DWORD_1 := dwArm1VertStn9SpSlanted); // CMP_OC_DW
ARdwVert4StepsPos_In_PositioningEn[1].20 := Stn9VertSlowPulldown.BZ_OUTPUT_BOOL;
AR3s_Vert4Steps_bTargetPosSt[1,9,2] := Stn9VertSlowPulldown.BZ_OUTPUT_BOOL;

END_PROGRAM

(* stored: Version 1.1.0.1, ProductVersion 3.1.4024.12
   POU AxisVertMovementOutputCtrl_Arm1: Id {2724bdc1-02a1-4d90-a283-50b987589666}, SpecialFunc None *)
